PROGRAM Gate_Small_Move
VAR
	smallGateGearIn				:MC_GearIn;				// 小龙门电子齿轮，LeftAxis为Master
	smallGateGearOut			:MC_GearOut;			// 小龙门电子齿轮取消啮合
	smallGateLeftAxisJog		:MC_Jog;				// 小龙门左轴(电子齿轮的Master轴)MC_Jog
	smallGateLeftAxisMoveAbs	:MC_MoveAbsolute;		// 小龙门MoveAbs(实际上电子齿轮的Master轴axis_SmallGate_Left的Mc_MoveAbsolute)
	
	// 默认为啮合状态，当激活大龙门左轴或者右轴的手动控制时bManualCtrl_Part_SmallGate_Left为true
	//或bManualCtrl_Part_SmallGate_Right为True，会把此变量置false
	bSmallGate_Gearin_do		:BOOL:=TRUE;
	
	nSmallGate_Speed					:LREAL:=2;		// 小龙门移动速度
	nSmallGate_MoveAbs_TarPos			:LREAL;			// 小龙门MoveAbs目标位置
	
END_VAR

// SmallGate Mc_Jog
smallGateLeftAxisJog(
	Axis:= axis_SmallGate_Left, 
	JogForward:= bSmallGate_Up, 
	JogBackwards:= bSmallGate_Down, 
	Mode:= MC_JOGMODE_CONTINOUS, 
	Position:= , 
	Velocity:= nSmallGate_Speed, 
	Acceleration:= , 
	Deceleration:= , 
	Jerk:= , 
	Done=> , 
	Busy=> , 
	Active=> , 
	CommandAborted=> , 
	Error=> , 
	ErrorID=> );

// SmallGate Mc_MoveAbsolute
smallGateLeftAxisMoveAbs(
	Axis:= axis_SmallGate_Left, 
	Execute:= bSmallGate_MoveAbs, 
	Position:= nSmallGate_MoveAbs_TarPos, 
	Velocity:= nSmallGate_Speed, 
	Acceleration:= , 
	Deceleration:= , 
	Jerk:= , 
	BufferMode:= , 
	Options:= , 
	Done=> , 
	Busy=> , 
	Active=> , 
	CommandAborted=> , 
	Error=> , 
	ErrorID=> );
	
smallGateGearIn(
	Master:= axis_SmallGate_Left, 
	Slave:= axis_SmallGate_Right, 
	Execute:= bSmallGate_Gearin_do, 
	RatioNumerator:= -1, 
	RatioDenominator:= 1, 
	Acceleration:= , 
	Deceleration:= , 
	Jerk:= , 
	BufferMode:= , 
	Options:= , 
	InGear=> , 
	Busy=> , 
	Active=> , 
	CommandAborted=> , 
	Error=> , 
	ErrorID=> );
	
	
smallGateGearOut(
	Slave:= axis_SmallGate_Right, 
	Execute:= NOT bSmallGate_Gearin_do, 
	Options:= , 
	Done=> , 
	Busy=> , 
	Error=> , 
	ErrorID=> );

END_PROGRAM

(* stored: Version 1.1.0.1, ProductVersion 3.1.4024.14
   POU Gate_Small_Move: Id {88f5fbeb-adda-460e-b025-9b481bebc10d}, SpecialFunc None *)
